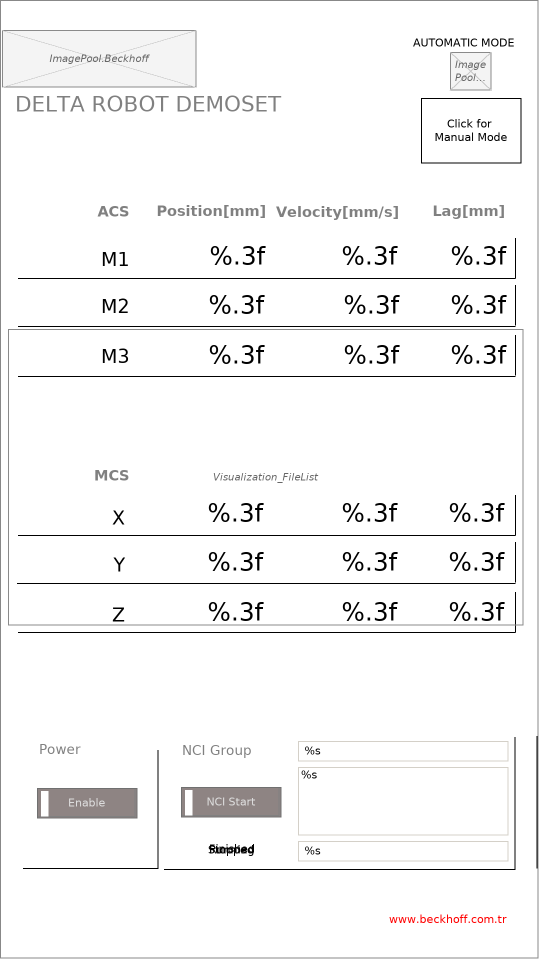
VISUALIZATION Visualization_AxesInfo  // 539x959, background image ImagePool.Background
    Label (35,229 155x61), "M1"
    Textfield (148,231 120x50), "%.3f", text variable: GVL_Axis.AxisM1_B.NcToPlc.ActPos
    Rectangle (39,248 7x22), invisible if: not stAxisM1_B.Out.xEnabled
    Rectangle (27,248 7x22), invisible if: not stAxisM1_B.Out.xAxisError
    Label (11,183 122x57), "ACS"
    Textfield (280,231 120x50), "%.3f", text variable: GVL_Axis.AxisM1_B.NcToPlc.ActVelo
    Image (2,30 194x57), image: ImagePool.Beckhoff
    Textfield (389,231 120x50), "%.3f", text variable: GVL_Axis.AxisM1_B.NcToPlc.PosDiff
    Line (18,278) (515,278)
    Line (515,238) (515,278)
    Label (38,276 155x61), "M2"
    Textfield (147,280 120x50), "%.3f", text variable: GVL_Axis.AxisM2_C.NcToPlc.ActPos
    Rectangle (39,295 7x22), invisible if: not stAxisM2_C.Out.xEnabled
    Rectangle (27,295 7x22), invisible if: not stAxisM2_C.Out.xAxisError
    Textfield (282,280 120x50), "%.3f", text variable: GVL_Axis.AxisM2_C.NcToPlc.ActVelo
    Textfield (389,280 120x50), "%.3f", text variable: GVL_Axis.AxisM2_C.NcToPlc.PosDiff
    Line (515,285) (515,325)
    Label (38,326 155x61), "M3"
    Textfield (147,330 120x50), "%.3f", text variable: GVL_Axis.AxisM3_A.NcToPlc.ActPos
    Rectangle (39,345 7x22), invisible if: not stAxisM3_A.Out.xEnabled
    Rectangle (27,345 7x22), invisible if: not stAxisM3_A.Out.xAxisError
    Textfield (282,330 120x50), "%.3f", text variable: GVL_Axis.AxisM3_A.NcToPlc.ActVelo
    Textfield (389,330 120x50), "%.3f", text variable: GVL_Axis.AxisM3_A.NcToPlc.PosDiff
    Line (18,376) (515,376)
    Line (515,335) (515,375)
    Line (18,326) (515,326)
    Label (11,447 122x57), "MCS"
    Label (8,493 120x50), "X"
    Textfield (126,488 140x50), "%.3f", text variable: GVL_Axis.AxisX.NcToPlc.ActPos
    Rectangle (39,505 7x22), invisible if: not stAxisX.Out.xEnabled
    Rectangle (27,505 7x22), invisible if: not stAxisX.Out.xAxisError
    Textfield (280,488 120x50), "%.3f", text variable: GVL_Axis.AxisX.NcToPlc.ActVelo
    Textfield (387,488 120x50), "%.3f", text variable: GVL_Axis.AxisX.NcToPlc.PosDiff
    Line (18,535) (515,535)
    Line (515,495) (515,535)
    Label (8,540 120x50), "Y"
    Textfield (126,537 140x50), "%.3f", text variable: GVL_Axis.AxisY.NcToPlc.ActPos
    Rectangle (39,552 7x22), invisible if: not stAxisY.Out.xEnabled
    Rectangle (27,552 6x22), invisible if: not stAxisY.Out.xAxisError
    Textfield (280,537 120x50), "%.3f", text variable: GVL_Axis.AxisY.NcToPlc.ActVelo
    Textfield (387,537 120x50), "%.3f", text variable: GVL_Axis.AxisY.NcToPlc.PosDiff
    Line (515,542) (515,582)
    Label (8,590 120x50), "Z"
    Textfield (126,587 140x50), "%.3f", text variable: GVL_Axis.AxisZ.NcToPlc.ActPos
    Rectangle (39,602 7x22), invisible if: not stAxisZ.Out.xEnabled
    Rectangle (27,602 7x22), invisible if: not stAxisZ.Out.xAxisError
    Textfield (280,587 120x50), "%.3f", text variable: GVL_Axis.AxisZ.NcToPlc.ActVelo
    Textfield (387,587 120x50), "%.3f", text variable: GVL_Axis.AxisZ.NcToPlc.PosDiff
    Line (18,632) (515,632)
    Line (515,592) (515,632)
    Line (17,583) (515,583)
    Textfield (298,767 210x68), "%s", text variable: PRG_NcControl.sNciLines
    Textfield (298,741 210x20), "%s", text variable: PRG_NcControl.sNciActualLine
    Label (189,834 86x30), "Finished", invisible if: NOT PRG_NcControl.bProgramFinished
    Label (188,835 86x30), "Stopped", invisible if: NOT PRG_NcControl.bProgramStopped
    Label (189,835 86x30), "Running", invisible if: NOT PRG_NcControl.bProgramRunning or PRG_NcControl.bProgramStopped
    Button (181,787 100x30), "NCI Start"
        toggle GVL_Process.bNciStartPLC
    Rectangle (185,790 7x25), invisible if: not PRG_NcControl.bNciStart
    Line (164,869) (515,869)
    Line (537,868) (537,736), invisible if: PRG_Process.bInvisible
    Label (147,722 140x57), "NCI Group"
    Textfield (298,841 210x20), "%s", text variable: PRG_Process.sFileNameVisu, input disabled if: PRG_NcControl.bProgramRunning
        toggle PRG_Process.bChangeFile
    Image (450,52 41x38), image: ImagePool.Mode_icon
        OnMouseMove: execute { GVL_Process.bMessageBubbleAuto := 1; }
        OnMouseClick: change screen: Visualization_AxesInfo_Manual
        OnMouseLeave: execute { GVL_Process.bMessageBubbleAuto := false; }
    Label (404,29 120x28), "AUTOMATIC MODE"
    Rectangle (421,98 100x65), "Click for Manual Mode", invisible if: not GVL_Process.bMessageBubbleAuto
    Frame (8,329 515x296), invisible if: not PRG_Process.bChangeFile
        shows Visualization_FileList()
    Label (12,77 308x54), "DELTA ROBOT DEMOSET"
    Label (149,186 120x50), "Position[mm]"
    Label (276,187 126x50), "Velocity[mm/s]"
    Label (388,186 120x50), "Lag[mm]"
    Button (37,788 100x30), "Enable"
        toggle GVL_Process.bAllAxesEnablePLC
    Rectangle (41,791 7x25), invisible if: not GVL_Process.bAllAxesEnable
    Line (23,868) (158,868)
    Line (158,868) (158,750)
    Label (25,721 70x57), "Power"
    Label (373,882 150x75), "www.beckhoff.com.tr"
    Line (515,869) (515,737)
END_VISUALIZATION

(* stored: Version 1.1.0.1, ProductVersion 3.1.4022.6
   Visu Visualization_AxesInfo: Id {3fde6272-4a97-451a-b04d-92f1e7932ca5} *)
